Staubli VAL3: init.pgx

program init(num x_nEncNum, string x_sTask)
begin
  //
  //***************************
  //***** Numerical value *****
  //***************************
  nPresetPos=0
  // -- Max value of module 750-631 encoder input in counts:
  // internal counter is unsigned 16 bits
  nMAXCOUNT=power(2,16)
  nMINCOUNT=0
  //
  //***************************
  //********* Strings *********
  //***************************
  sTASK=x_sTask+toString("",x_nEncNum)
  sEncNum="ENC"+toString("",x_nEncNum)
  //
  //***************************
  //* INITIALIZATION  SECTION *
  //***************************
  //-- Detection of rising edge on encoder latch input
  bMemoLatchState=diEncLatched
  //-- Part has been latched
  bPartLatched=false
  //
  // Preset encoder counter
  aioSet(aoPresetPos,nPresetPos)
  doEnablePreset=true
  //
  // Reset latch register
  doEnableLatch=false
  //
  //-- Get value Overflow/Underflow status bit
  //   to detect rising edges
  bMemoOvf=diOverFlow
  bMemoUdf=diUnderFlow
  //
  // Initialize encoder values
  nEncLatchedVal=nEncValue=0
  //
  bLatchEnabled=true
end
